(* PLC project CoDeSys External Library Template, WAGO e!COCKPIT e!COCKPIT, author 3S - Smart Software Solutions GmbH *)
(* stored: creationDateTime 2019-10-29T12:37:19.5105513, version 3.5.5.30, modificationDateTime 2019-10-29T12:36:39.3744516, organization 3S - Smart Software Solutions GmbH *)
(* Library project template with all possible element types, docu and a sample project structure *)

TYPE SILOWNIK_HRU : STRUCT
  sIdInstancji : STRING;
  intTrybPracy : INT;
  xBrakKomunikacjiIZE : BOOL;
  xBrakKomunikacjiPLC : BOOL;
  xPokazPanelHMI : BOOL := TRUE;
  rTemperaturaPomieszczenia : REAL;
  rNastawaPolozeniaSilownika : REAL;
  rZadanePolozenieSilownikaHMI : REAL;
  intTrybPracyHMI : INT := 1;
  xAutonomizacja : BOOL;
  xAlarmOgolny : BOOL;
  xBladBaterii : BOOL;
  xDetekcjaOtwarciaOkna : BOOL;
  sEnOceanIDodczytany : STRING;
  wCzasOdOstatniegoKomunikatu : WORD;
  xPoprawneParowanie : BOOL;
  xUczenieWlaczHMI : BOOL;
  xUczenieWlaczone : BOOL;
  xUsuwaniePotwierdzenieHMI : BOOL;
  xUsuwanieHMI : BOOL;
END_STRUCT;
END_TYPE
